# EPICS substitutions: pmacUtilApp/Db/geobrickette_motion_stop.substitutions
file motion_protection.template
{
pattern {P,    PORT }
        {$(P), $(PORT)}
}

file motion_protection.template
{
pattern {P,    Q,                    PORT,    DESC,               , VAR, ZNAM,         ZSV,   ONAM,     OSV}
        {$(P), ":MOTIONSTOP_ACTIVE", $(PORT), "motion stop active", I35, "Not Active", MINOR, "Active", NO_ALARM }
}
